Staubli VAL3: refresh.pgx

program refresh()
// // page refresh
begin
  // refresh the static message
  if !bShowStatus
    if (nKey>=270 and nKey<=278) or use:bUseRefresh
      call refreshStatic()
      call refreshDynamic()
    else
      if !bShowStatus
        // refresh the Dynamic message
        if (clock()-nRefresh>nTime)
          call refreshDynamic()
        endIf
      endIf
    endIf
  endIf
  // show the coordinate
  call showStatus()
  // release the resource
  delay(0)
end
